// TIA Portal project "测试项目程序1500" (V18)

(* hardware
DEVICE "S7-1500/ET200MP station_1"  S7-1500 station
   slot 0: "导轨_0"  Rack  6ES7 590-1***0-0AA0
   slot 1: "PLC_1"  CPU 1513-1 PN  6ES7 513-1AL02-0AB0  V2.9
      slot 3: "CPU 显示_1"  6ES7591-1AA00-0AA0
      slot 32768: "PROFINET 接口_1"  X1
         slot 32769: "端口_1"  X1 P1
         slot 32770: "端口_2"  X1 P2
      slot 34817: "Virtual CP interface port_1"  Virtual CP interface port  Virtual CP interface port
*)

// ===== PLC "PLC_1"  CPU 1513-1 PN =====

VAR_GLOBAL   // PLC tag table "默认变量表"
   "FirstScan" AT %M1.0 : Bool;
   "DiagStatusUpdate" AT %M1.1 : Bool;
   "AlwaysTRUE" AT %M1.2 : Bool;
   "AlwaysFALSE" AT %M1.3 : Bool;
   "System_Byte" AT %MB1 : Byte;
   "Clock_Byte" AT %MB0 : Byte;
   "Clock_10Hz" AT %M0.0 : Bool;
   "Clock_5Hz" AT %M0.1 : Bool;
   "Clock_2.5Hz" AT %M0.2 : Bool;
   "Clock_2Hz" AT %M0.3 : Bool;
   "Clock_1.25Hz" AT %M0.4 : Bool;
   "Clock_1Hz" AT %M0.5 : Bool;
   "Clock_0.625Hz" AT %M0.6 : Bool;
   "Clock_0.5Hz" AT %M0.7 : Bool;
   "Tag_1" AT %IW0 : Int;
   "Tag_2" AT %IW2 : Int;
   "Tag_3" AT %IW4 : Int;
   "Tag_4" AT %IW6 : Int;
   "Tag_5" AT %IW8 : Int;
   "Tag_6" AT %IW10 : Int;
   "Tag_7" AT %IW12 : Int;
   "Tag_8" AT %IW14 : Int;
   "Tag_9" AT %IW16 : Int;
END_VAR

DATA_BLOCK "控制设定"   // DB1
{ S7_Optimized_Access := 'FALSE' }
VERSION : 0.1
   VAR
      进水泵状态 : Bool;
      加水泵状态 : Bool;
      燃气泵状态 : Bool;
      循环泵状态 : Bool;
      出水阀状态 : Bool;
      系统状态 : Bool;
      系统状态_1 : Bool;
      系统状态_2 : Bool;
      系统状态_3 : Bool;
      系统状态_4 : Bool;
      系统状态_5 : Bool;
      系统状态_6 : Bool;
      系统状态_7 : Bool;
      系统状态_8 : Bool;
      系统状态_9 : Bool;
      系统状态_10 : Bool;
      系统状态_11 : Bool;
      进水压力 : Real;
      出水压力 : Real;
      进水温度 : Real;
      出水温度 : Real;
      水罐液位 : Real;
      锅炉液位 : Real;
      锅炉温度 : Real;
      锅炉压力 : Real;
      管道流动压力 : Real;
      备用2 : Real;
      备用3 : Real;
      备用4 : Real;
      备用5 : Real;
      备用6 : Real;
      备用7 : Real;
      备用8 : Real;
      备用9 : Real;
      备用10 : Real;
      备用11 : Real;
      备用12 : Real;
      备用13 : Real;
      备用14 : Real;
      备用15 : Real;
      备用16 : Int;
      备用17 : Int;
      进水泵启动 : Bool;
      进水泵停止 : Bool;
      加水泵启动 : Bool;
      加水泵停止 : Bool;
      燃气泵启动 : Bool;
      燃气泵停止 : Bool;
      循环泵启动 : Bool;
      循环泵停止 : Bool;
      出水阀启动 : Bool;
      出水阀停止 : Bool;
      PLC上位机信号开 : Bool;
      PLC上位机信号关 : Bool;
   END_VAR
BEGIN
END_DATA_BLOCK

DATA_BLOCK "模拟量数据"   // DB2
{ S7_Optimized_Access := 'FALSE' }
VERSION : 0.1
   VAR
      启动 : Bool;
      停止 : Bool;
      故障复位 : Bool;
      热保护 : Bool;
      故障指示灯 : Bool;
      设定时间 : Time;
      当前时间 : Time;
      电机 : Bool;
      定时器 : IEC_TIMER;
      频率反馈 : Real;
      断线报警 : Bool;
      超限报警 : Bool;
      频率给定 : Real;
      断线报警1 : Bool;
      超限报警1 : Bool;
   END_VAR
BEGIN
END_DATA_BLOCK

FUNCTION "泵_控制" : Void   // FC1, LAD
{ S7_Optimized_Access := 'TRUE' }
VERSION : 0.1
BEGIN

REGION Network 1: 进水泵
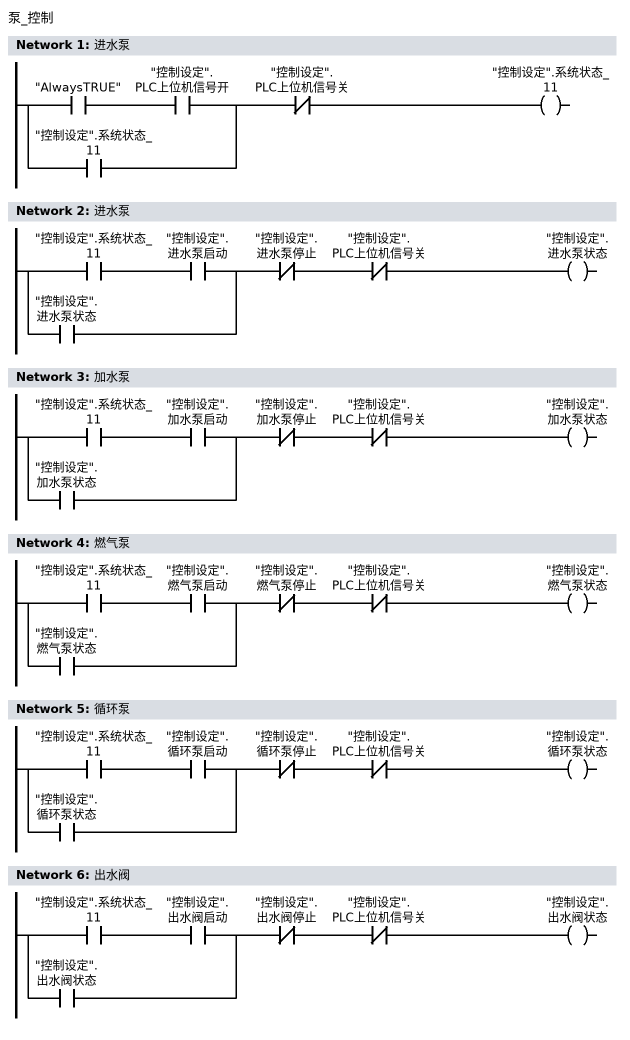
   RUNG wire#powerrail
      Contact( "AlwaysTRUE" )
      Contact( "控制设定".PLC上位机信号开 )
      wire#w1
      I_Contact( "控制设定".PLC上位机信号关 )
      Coil( "控制设定".系统状态_11 )
   END_RUNG
   RUNG wire#powerrail
      Contact( "控制设定".系统状态_11 )
   END_RUNG wire#w1
   // the same network as SCL:
   "控制设定".系统状态_11 := (("AlwaysTRUE" AND "控制设定".PLC上位机信号开) OR "控制设定".系统状态_11) AND NOT "控制设定".PLC上位机信号关;
END_REGION

REGION Network 2: 进水泵
   RUNG wire#powerrail
      Contact( "控制设定".系统状态_11 )
      Contact( "控制设定".进水泵启动 )
      wire#w1
      I_Contact( "控制设定".进水泵停止 )
      I_Contact( "控制设定".PLC上位机信号关 )
      Coil( "控制设定".进水泵状态 )
   END_RUNG
   RUNG wire#powerrail
      Contact( "控制设定".进水泵状态 )
   END_RUNG wire#w1
   // the same network as SCL:
   "控制设定".进水泵状态 := (("控制设定".系统状态_11 AND "控制设定".进水泵启动) OR "控制设定".进水泵状态) AND NOT "控制设定".进水泵停止 AND NOT "控制设定".PLC上位机信号关;
END_REGION

REGION Network 3: 加水泵
   RUNG wire#powerrail
      Contact( "控制设定".系统状态_11 )
      Contact( "控制设定".加水泵启动 )
      wire#w1
      I_Contact( "控制设定".加水泵停止 )
      I_Contact( "控制设定".PLC上位机信号关 )
      Coil( "控制设定".加水泵状态 )
   END_RUNG
   RUNG wire#powerrail
      Contact( "控制设定".加水泵状态 )
   END_RUNG wire#w1
   // the same network as SCL:
   "控制设定".加水泵状态 := (("控制设定".系统状态_11 AND "控制设定".加水泵启动) OR "控制设定".加水泵状态) AND NOT "控制设定".加水泵停止 AND NOT "控制设定".PLC上位机信号关;
END_REGION

REGION Network 4: 燃气泵
   RUNG wire#powerrail
      Contact( "控制设定".系统状态_11 )
      Contact( "控制设定".燃气泵启动 )
      wire#w1
      I_Contact( "控制设定".燃气泵停止 )
      I_Contact( "控制设定".PLC上位机信号关 )
      Coil( "控制设定".燃气泵状态 )
   END_RUNG
   RUNG wire#powerrail
      Contact( "控制设定".燃气泵状态 )
   END_RUNG wire#w1
   // the same network as SCL:
   "控制设定".燃气泵状态 := (("控制设定".系统状态_11 AND "控制设定".燃气泵启动) OR "控制设定".燃气泵状态) AND NOT "控制设定".燃气泵停止 AND NOT "控制设定".PLC上位机信号关;
END_REGION

REGION Network 5: 循环泵
   RUNG wire#powerrail
      Contact( "控制设定".系统状态_11 )
      Contact( "控制设定".循环泵启动 )
      wire#w1
      I_Contact( "控制设定".循环泵停止 )
      I_Contact( "控制设定".PLC上位机信号关 )
      Coil( "控制设定".循环泵状态 )
   END_RUNG
   RUNG wire#powerrail
      Contact( "控制设定".循环泵状态 )
   END_RUNG wire#w1
   // the same network as SCL:
   "控制设定".循环泵状态 := (("控制设定".系统状态_11 AND "控制设定".循环泵启动) OR "控制设定".循环泵状态) AND NOT "控制设定".循环泵停止 AND NOT "控制设定".PLC上位机信号关;
END_REGION

REGION Network 6: 出水阀
   RUNG wire#powerrail
      Contact( "控制设定".系统状态_11 )
      Contact( "控制设定".出水阀启动 )
      wire#w1
      I_Contact( "控制设定".出水阀停止 )
      I_Contact( "控制设定".PLC上位机信号关 )
      Coil( "控制设定".出水阀状态 )
   END_RUNG
   RUNG wire#powerrail
      Contact( "控制设定".出水阀状态 )
   END_RUNG wire#w1
   // the same network as SCL:
   "控制设定".出水阀状态 := (("控制设定".系统状态_11 AND "控制设定".出水阀启动) OR "控制设定".出水阀状态) AND NOT "控制设定".出水阀停止 AND NOT "控制设定".PLC上位机信号关;
END_REGION
END_FUNCTION

FUNCTION "模拟量_采集" : Void   // FC2, LAD
{ S7_Optimized_Access := 'TRUE' }
VERSION : 0.1
   VAR_INPUT
      模拟量输入 : Int;
      模拟量上限 : Int;
      模拟量下限 : Int;
      量程上限 : Real;
      量程下限 : Real;
   END_VAR
   VAR_OUTPUT
      实际值 : Real;
      断线报警 : Bool;
      超限报警 : Bool;
   END_VAR
   VAR_TEMP
      过程值 : Real;
   END_VAR
BEGIN

REGION Network 1
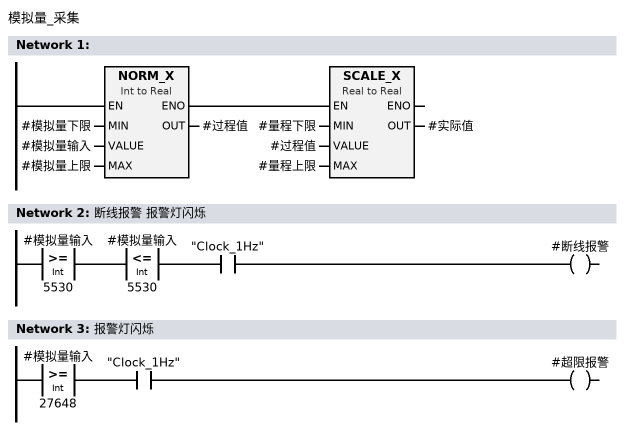
   RUNG wire#powerrail
      { S7_Templates := "[SrcType := Int, DestType := Real]" } Normalize(min := #模拟量下限, value := #模拟量输入, max := #模拟量上限, out => #过程值)
      { S7_Templates := "[SrcType := Real, DestType := Real]" } Scale(min := #量程下限, value := #过程值, max := #量程上限, out => #实际值)
   END_RUNG
   // the same network as SCL:
   #过程值 := NORM_X(MIN := #模拟量下限, VALUE := #模拟量输入, MAX := #模拟量上限);
   #实际值 := SCALE_X(MIN := #量程下限, VALUE := #过程值, MAX := #量程上限);
END_REGION

REGION Network 2: 断线报警 报警灯闪烁
   RUNG wire#powerrail
      { S7_Templates := "SrcType := Int" } GE_Contact(in1 := #模拟量输入, in2 := 5530)
      { S7_Templates := "SrcType := Int" } LE_Contact(in1 := #模拟量输入, in2 := 5530)
      Contact( "Clock_1Hz" )
      Coil( #断线报警 )
   END_RUNG
   // the same network as SCL:
   #断线报警 := (#模拟量输入 >= 5530) AND (#模拟量输入 <= 5530) AND "Clock_1Hz";
END_REGION

REGION Network 3: 报警灯闪烁
   RUNG wire#powerrail
      { S7_Templates := "SrcType := Int" } GE_Contact(in1 := #模拟量输入, in2 := 27648)
      Contact( "Clock_1Hz" )
      Coil( #超限报警 )
   END_RUNG
   // the same network as SCL:
   #超限报警 := (#模拟量输入 >= 27648) AND "Clock_1Hz";
END_REGION
END_FUNCTION

FUNCTION "模拟量_设定" : Void   // FC3, LAD
{ S7_Optimized_Access := 'TRUE' }
VERSION : 0.1
   VAR_INPUT
      模拟量输入 : Real;
      量程上限 : Real;
      量程下限 : Real;
      模拟量上限 : Int;
      模拟量下限 : Int;
   END_VAR
   VAR_OUTPUT
      给定值 : Int;
      断线报警 : Bool;
      超限报警 : Bool;
   END_VAR
   VAR_TEMP
      过程值 : Real;
   END_VAR
BEGIN

REGION Network 1: 频率给定
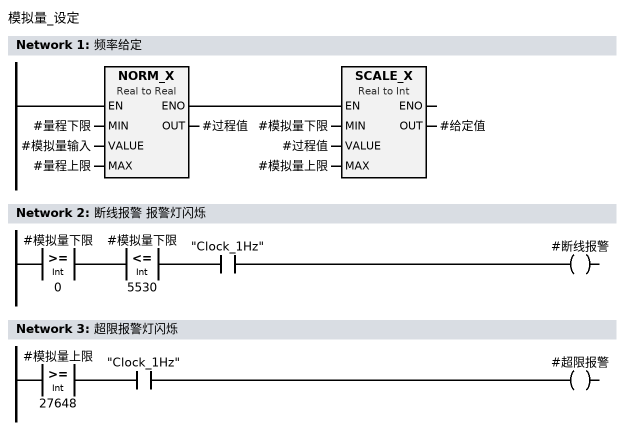
   RUNG wire#powerrail
      { S7_Templates := "[SrcType := Real, DestType := Real]" } Normalize(min := #量程下限, value := #模拟量输入, max := #量程上限, out => #过程值)
      { S7_Templates := "[SrcType := Real, DestType := Int]" } Scale(min := #模拟量下限, value := #过程值, max := #模拟量上限, out => #给定值)
   END_RUNG
   // the same network as SCL:
   #过程值 := NORM_X(MIN := #量程下限, VALUE := #模拟量输入, MAX := #量程上限);
   #给定值 := SCALE_X(MIN := #模拟量下限, VALUE := #过程值, MAX := #模拟量上限);
END_REGION

REGION Network 2: 断线报警 报警灯闪烁
   RUNG wire#powerrail
      { S7_Templates := "SrcType := Int" } GE_Contact(in1 := #模拟量下限, in2 := 0)
      { S7_Templates := "SrcType := Int" } LE_Contact(in1 := #模拟量下限, in2 := 5530)
      Contact( "Clock_1Hz" )
      Coil( #断线报警 )
   END_RUNG
   // the same network as SCL:
   #断线报警 := (#模拟量下限 >= 0) AND (#模拟量下限 <= 5530) AND "Clock_1Hz";
END_REGION

REGION Network 3: 超限报警灯闪烁
   RUNG wire#powerrail
      { S7_Templates := "SrcType := Int" } GE_Contact(in1 := #模拟量上限, in2 := 27648)
      Contact( "Clock_1Hz" )
      Coil( #超限报警 )
   END_RUNG
   // the same network as SCL:
   #超限报警 := (#模拟量上限 >= 27648) AND "Clock_1Hz";
END_REGION
END_FUNCTION

FUNCTION "模拟量" : Void   // FC4, LAD
{ S7_Optimized_Access := 'TRUE' }
VERSION : 0.1
   VAR_TEMP   // added for the SCL form of the ladder/FBD networks
      _w1 : Bool;
   END_VAR
BEGIN

REGION Network 1
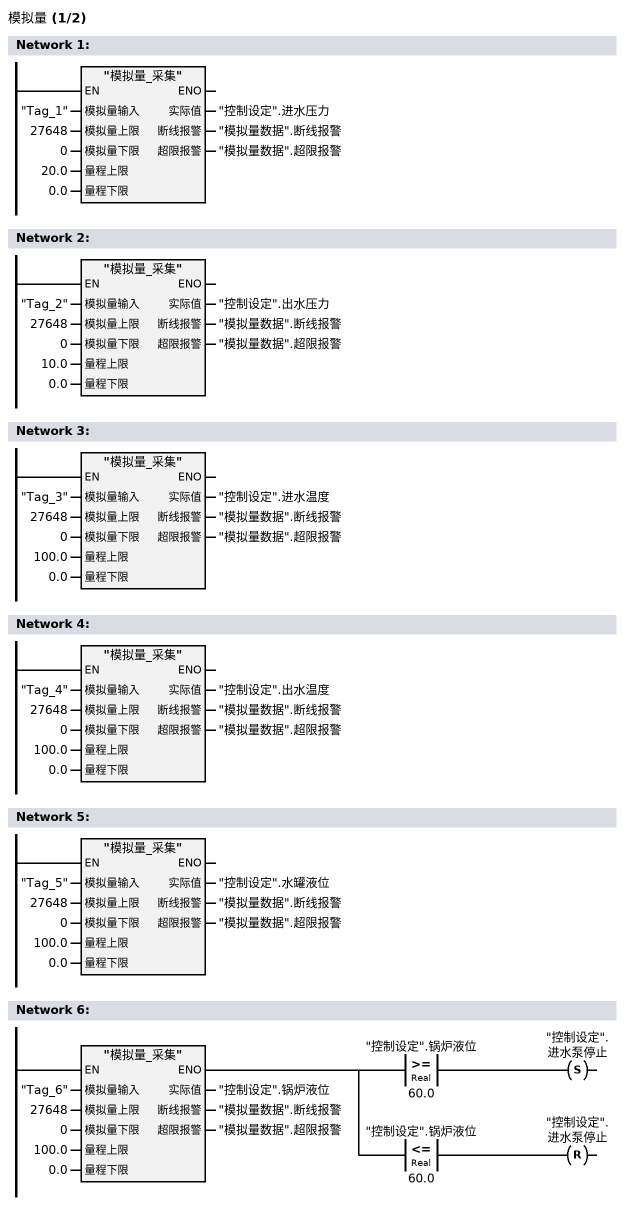
   RUNG wire#powerrail
      "模拟量_采集"(模拟量输入 := "Tag_1", 模拟量上限 := 27648, 模拟量下限 := 0, 量程上限 := 20.0, 量程下限 := 0.0, 实际值 => "控制设定".进水压力, 断线报警 => "模拟量数据".断线报警, 超限报警 => "模拟量数据".超限报警)
   END_RUNG
   // the same network as SCL:
   "模拟量_采集"(模拟量输入 := "Tag_1",
            模拟量上限 := 27648,
            模拟量下限 := 0,
            量程上限 := 20.0,
            量程下限 := 0.0,
            实际值 => "控制设定".进水压力,
            断线报警 => "模拟量数据".断线报警,
            超限报警 => "模拟量数据".超限报警);
END_REGION

REGION Network 2
   RUNG wire#powerrail
      "模拟量_采集"(模拟量输入 := "Tag_2", 模拟量上限 := 27648, 模拟量下限 := 0, 量程上限 := 10.0, 量程下限 := 0.0, 实际值 => "控制设定".出水压力, 断线报警 => "模拟量数据".断线报警, 超限报警 => "模拟量数据".超限报警)
   END_RUNG
   // the same network as SCL:
   "模拟量_采集"(模拟量输入 := "Tag_2",
            模拟量上限 := 27648,
            模拟量下限 := 0,
            量程上限 := 10.0,
            量程下限 := 0.0,
            实际值 => "控制设定".出水压力,
            断线报警 => "模拟量数据".断线报警,
            超限报警 => "模拟量数据".超限报警);
END_REGION

REGION Network 3
   RUNG wire#powerrail
      "模拟量_采集"(模拟量输入 := "Tag_3", 模拟量上限 := 27648, 模拟量下限 := 0, 量程上限 := 100.0, 量程下限 := 0.0, 实际值 => "控制设定".进水温度, 断线报警 => "模拟量数据".断线报警, 超限报警 => "模拟量数据".超限报警)
   END_RUNG
   // the same network as SCL:
   "模拟量_采集"(模拟量输入 := "Tag_3",
            模拟量上限 := 27648,
            模拟量下限 := 0,
            量程上限 := 100.0,
            量程下限 := 0.0,
            实际值 => "控制设定".进水温度,
            断线报警 => "模拟量数据".断线报警,
            超限报警 => "模拟量数据".超限报警);
END_REGION

REGION Network 4
   RUNG wire#powerrail
      "模拟量_采集"(模拟量输入 := "Tag_4", 模拟量上限 := 27648, 模拟量下限 := 0, 量程上限 := 100.0, 量程下限 := 0.0, 实际值 => "控制设定".出水温度, 断线报警 => "模拟量数据".断线报警, 超限报警 => "模拟量数据".超限报警)
   END_RUNG
   // the same network as SCL:
   "模拟量_采集"(模拟量输入 := "Tag_4",
            模拟量上限 := 27648,
            模拟量下限 := 0,
            量程上限 := 100.0,
            量程下限 := 0.0,
            实际值 => "控制设定".出水温度,
            断线报警 => "模拟量数据".断线报警,
            超限报警 => "模拟量数据".超限报警);
END_REGION

REGION Network 5
   RUNG wire#powerrail
      "模拟量_采集"(模拟量输入 := "Tag_5", 模拟量上限 := 27648, 模拟量下限 := 0, 量程上限 := 100.0, 量程下限 := 0.0, 实际值 => "控制设定".水罐液位, 断线报警 => "模拟量数据".断线报警, 超限报警 => "模拟量数据".超限报警)
   END_RUNG
   // the same network as SCL:
   "模拟量_采集"(模拟量输入 := "Tag_5",
            模拟量上限 := 27648,
            模拟量下限 := 0,
            量程上限 := 100.0,
            量程下限 := 0.0,
            实际值 => "控制设定".水罐液位,
            断线报警 => "模拟量数据".断线报警,
            超限报警 => "模拟量数据".超限报警);
END_REGION

REGION Network 6
   RUNG wire#powerrail
      "模拟量_采集"(模拟量输入 := "Tag_6", 模拟量上限 := 27648, 模拟量下限 := 0, 量程上限 := 100.0, 量程下限 := 0.0, 实际值 => "控制设定".锅炉液位, 断线报警 => "模拟量数据".断线报警, 超限报警 => "模拟量数据".超限报警)
      wire#w1
      { S7_Templates := "SrcType := Real" } GE_Contact(in1 := "控制设定".锅炉液位, in2 := 60.0)
      S_Coil( "控制设定".进水泵停止 )
   END_RUNG
   RUNG wire#w1
      { S7_Templates := "SrcType := Real" } LE_Contact(in1 := "控制设定".锅炉液位, in2 := 60.0)
      R_Coil( "控制设定".进水泵停止 )
   END_RUNG
   // the same network as SCL:
   "模拟量_采集"(模拟量输入 := "Tag_6",
            模拟量上限 := 27648,
            模拟量下限 := 0,
            量程上限 := 100.0,
            量程下限 := 0.0,
            实际值 => "控制设定".锅炉液位,
            断线报警 => "模拟量数据".断线报警,
            超限报警 => "模拟量数据".超限报警,
            ENO => #_w1);
   IF #_w1 AND ("控制设定".锅炉液位 >= 60.0) THEN "控制设定".进水泵停止 := TRUE; END_IF;
   IF #_w1 AND ("控制设定".锅炉液位 <= 60.0) THEN "控制设定".进水泵停止 := FALSE; END_IF;
END_REGION

REGION Network 7
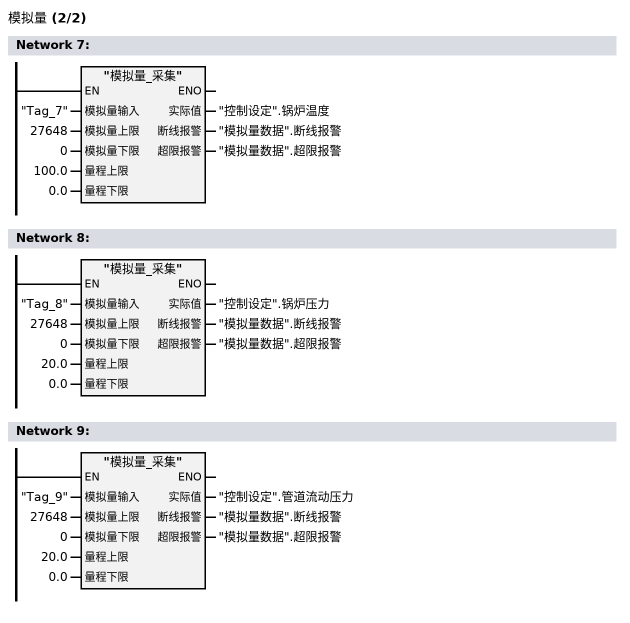
   RUNG wire#powerrail
      "模拟量_采集"(模拟量输入 := "Tag_7", 模拟量上限 := 27648, 模拟量下限 := 0, 量程上限 := 100.0, 量程下限 := 0.0, 实际值 => "控制设定".锅炉温度, 断线报警 => "模拟量数据".断线报警, 超限报警 => "模拟量数据".超限报警)
   END_RUNG
   // the same network as SCL:
   "模拟量_采集"(模拟量输入 := "Tag_7",
            模拟量上限 := 27648,
            模拟量下限 := 0,
            量程上限 := 100.0,
            量程下限 := 0.0,
            实际值 => "控制设定".锅炉温度,
            断线报警 => "模拟量数据".断线报警,
            超限报警 => "模拟量数据".超限报警);
END_REGION

REGION Network 8
   RUNG wire#powerrail
      "模拟量_采集"(模拟量输入 := "Tag_8", 模拟量上限 := 27648, 模拟量下限 := 0, 量程上限 := 20.0, 量程下限 := 0.0, 实际值 => "控制设定".锅炉压力, 断线报警 => "模拟量数据".断线报警, 超限报警 => "模拟量数据".超限报警)
   END_RUNG
   // the same network as SCL:
   "模拟量_采集"(模拟量输入 := "Tag_8",
            模拟量上限 := 27648,
            模拟量下限 := 0,
            量程上限 := 20.0,
            量程下限 := 0.0,
            实际值 => "控制设定".锅炉压力,
            断线报警 => "模拟量数据".断线报警,
            超限报警 => "模拟量数据".超限报警);
END_REGION

REGION Network 9
   RUNG wire#powerrail
      "模拟量_采集"(模拟量输入 := "Tag_9", 模拟量上限 := 27648, 模拟量下限 := 0, 量程上限 := 20.0, 量程下限 := 0.0, 实际值 => "控制设定".管道流动压力, 断线报警 => "模拟量数据".断线报警, 超限报警 => "模拟量数据".超限报警)
   END_RUNG
   // the same network as SCL:
   "模拟量_采集"(模拟量输入 := "Tag_9",
            模拟量上限 := 27648,
            模拟量下限 := 0,
            量程上限 := 20.0,
            量程下限 := 0.0,
            实际值 => "控制设定".管道流动压力,
            断线报警 => "模拟量数据".断线报警,
            超限报警 => "模拟量数据".超限报警);
END_REGION
END_FUNCTION

FUNCTION "调用泵" : Void   // FC5, LAD
{ S7_Optimized_Access := 'TRUE' }
VERSION : 0.1
   VAR_INPUT
      启动 : Bool;
      停止 : Bool;
      故障复位 : Bool;
      热保护 : Bool;
      延时时间 : Time;
   END_VAR
   VAR_OUTPUT
      当前时间 : Time;
   END_VAR
   VAR_IN_OUT
      故障指示灯 : Bool;
      定时器 : IEC_TIMER;
      电机_1 : Bool;
   END_VAR
BEGIN

REGION Network 1
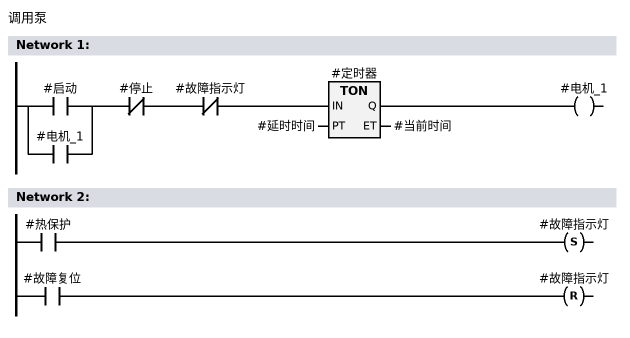
   #定时器.TON(IN := (#启动 OR #电机_1) AND NOT #停止 AND NOT #故障指示灯, PT := #延时时间, ET => #当前时间);
   #电机_1 := #定时器.Q;
END_REGION

REGION Network 2
   RUNG wire#powerrail
      Contact( #热保护 )
      S_Coil( #故障指示灯 )
   END_RUNG
   RUNG wire#powerrail
      Contact( #故障复位 )
      R_Coil( #故障指示灯 )
   END_RUNG
   // the same network as SCL:
   IF #热保护 THEN #故障指示灯 := TRUE; END_IF;
   IF #故障复位 THEN #故障指示灯 := FALSE; END_IF;
END_REGION
END_FUNCTION

ORGANIZATION_BLOCK "Main"   // OB1, LAD, ProgramCycle
TITLE = "Main Program Sweep (Cycle)"
{ S7_Optimized_Access := 'FALSE' }
VERSION : 0.1
   VAR_TEMP
      EV_CLASS : Byte;   // Bits 0-3 = 1:Coming event, Bits 4-7 = 1:Event class 1
      SCAN_1 : Byte;   // 1:Initial call of the OB, 3: Call 2-n of the OB
      PRIORITY : Byte;   // Priority of OB Execution
      OB_NUMBR : Byte;   // OB number
      RESERVED_1 : Byte;   // Reserved for system
      RESERVED_2 : Byte;   // Reserved for system
      PREV_CYCLE : Int;   // Previous program cycle time (milliseconds)
      MIN_CYCLE : Int;   // Minimum program cycle time (milliseconds)
      MAX_CYCLE : Int;   // Maximum program cycle time (milliseconds)
      DATE_TIME : Date_And_Time;   // Date and time OB started
   END_VAR
BEGIN

REGION Network 1
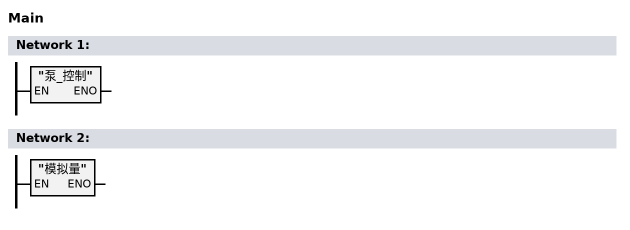
   RUNG wire#powerrail
      "泵_控制"()
   END_RUNG
   // the same network as SCL:
   "泵_控制"();
END_REGION

REGION Network 2
   RUNG wire#powerrail
      "模拟量"()
   END_RUNG
   // the same network as SCL:
   "模拟量"();
END_REGION
END_ORGANIZATION_BLOCK